PROGRAM P_Control
VAR
	fbControl1 : FB_Control;
	fbControl2 : FB_Control;
END_VAR

IF G_Enables.bAuto THEN
	
	fbControl1(
		fFF := G_OPC.fValveOneSignals.fFF,
		fPID := G_OPC.fValveOneSignals.fPID,
		fDeadBandUp := G_Parameters.fDeadUpOne,
		fDeadBandDown := G_Parameters.fDeadDownOne,
		fXDotRef := G_OPC.fXDotRefOne,
		fError := G_OPC.fValveOneSignals.fError,
		fKFF := G_Parameters.fOneMultiFF,

		bFF := G_Enables.bEnableFF,
		bPID := G_Enables.bEnablePID,
		bU := G_Enables.bEnableU, 
		
		fU => G_OPC.fValveOneSignals.fU
	);
	
	fbControl2(
		fFF := G_OPC.fValveTwoSignals.fFF,
		fPID := G_OPC.fValveTwoSignals.fPID,
		fDeadBandUp := G_Parameters.fDeadUpTwo,
		fDeadBandDown := G_Parameters.fDeadDownTwo,
		fXDotRef := G_OPC.fXDotRefTwo,
		fError := G_OPC.fValveTwoSignals.fError,
		fKFF := G_Parameters.fTwoMultiFF, 
		
		bFF := G_Enables.bEnableFF,
		bPID := G_Enables.bEnablePID,
		bU := G_Enables.bEnableU,
		
		fU => G_OPC.fValveTwoSignals.fU
	);
	
ELSIF G_Enables.bManSpeed THEN
	fbControl1(
		fFF := G_OPC.fValveOneSignals.fFF,
		fPID := G_OPC.fValveOneSignals.fPID,
		fDeadBandUp := G_Parameters.fDeadUpOne,
		fDeadBandDown := G_Parameters.fDeadDownOne,
		fXDotRef := G_OPC.fJoystickJib * G_Parameters.fMaxSpeedJib,
		fError := G_OPC.fValveOneSignals.fError,
		fKFF := G_Parameters.fOneMultiFF,

		bFF := G_Enables.bEnableFF,
		bPID := G_Enables.bEnablePID,
		bU := G_Enables.bEnableU, 
		
		fU => G_OPC.fValveOneSignals.fU
	);
	
	fbControl2(
		fFF := G_OPC.fValveTwoSignals.fFF,
		fPID := G_OPC.fValveTwoSignals.fPID,
		fDeadBandUp := G_Parameters.fDeadUpTwo,
		fDeadBandDown := G_Parameters.fDeadDownTwo,
		fXDotRef := G_OPC.fJoystickMain * G_Parameters.fMaxSpeedMain,
		fError := G_OPC.fValveTwoSignals.fError,
		fKFF := G_Parameters.fTwoMultiFF, 
		
		bFF := G_Enables.bEnableFF,
		bPID := G_Enables.bEnablePID,
		bU := G_Enables.bEnableU,
		
		fU => G_OPC.fValveTwoSignals.fU
	);
	
ELSE
	G_OPC.fValveOneSignals.fU := 0.0;
	G_OPC.fValveTwoSignals.fU := 0.0;
END_IF

END_PROGRAM

(* stored: Version 1.1.0.1
   POU P_Control: Id {97b90c20-1ebb-4d5f-92ff-63da301b4f7c}, SpecialFunc None *)
